PROGRAM P20_ErrorHandling
VAR
	GLOBAL_ERROR_STRING : STRING(200);
END_VAR


GLOBAL_ERROR_STRING := GVL_PLC.bGlobal_Error_String;

IF kidAxis.Status.Error THEN
	GVL_PLC.bGlobal_Error := TRUE;
	
END_IF

IF GVL_PLC.bGlobal_Reset THEN
	GLOBAL_ERROR_STRING := '';
	GVL_PLC.bGlobal_Error := FALSE;
	IF kidAxis.Status.Fault THEN
		GVL_Motion.bNC_Reset := TRUE;
		GVL_DriveParameters.controlWord := 128;
	END_IF

	GVL_PLC.bGlobal_Reset := FALSE;

END_IF

END_PROGRAM

(* stored: Version 1.1.0.1, ProductVersion 3.1.4022.3
   POU P20_ErrorHandling: Id {4160e03a-aba1-4f62-8d36-504ed33080ca}, SpecialFunc None *)
